{attribute 'qualified_only'}
{attribute 'to_string'}
TYPE ZAppStep :
(
  Undefined := 0
  
  ,BootBegin
  ,BootLoadDefaultData
  ,BootEnd
  ,BootFaultBegin
  ,BootFaultEnd 
  ,RunningBegin
  ,RunningEnd   
);
END_TYPE

(* stored: Version 1.1.0.1
   DUT ZAppStep: Id {29bbb3c0-58ec-4b84-8654-d7e4cc7534a1} *)
